Fanuc KAREL source: compact_preamble.KL

PROGRAM KA00132
%NOLOCKGROUP
VAR
SRC : ARRAY[2] OF BYTE
DST : ARRAY[2] OF SHORT
BEGIN
SRC[1]=2
DST[1]=SRC[1]
END KA00132
